INTERFACE I_HostOutputPorts EXTENDS __SYSTEM.IQueryInterface

METHOD PUBLIC AddDataAsOutputPort : I_OutputPort
VAR_INPUT
	Name : T_MAXSTRING;
	Data : I_Datatype;
END_VAR
END_METHOD

METHOD AddOutputPort
VAR_INPUT
	OutputPort : I_OutputPort;
END_VAR
END_METHOD

METHOD PUBLIC TryGetOutputPortByName : BOOL
VAR_INPUT
	Name : T_MAXSTRING;
	Destination : REFERENCE TO I_OutputPort;
END_VAR
END_METHOD

END_INTERFACE

(* stored: Version 1.1.0.1, ProductVersion 3.1.4024.12
   Itf I_HostOutputPorts: Id {5e1aea97-5e53-08af-11e9-4031292affee}
   Method AddDataAsOutputPort: Id {ae2495e6-ec41-49e7-bdb1-5ba1eea57cfd}
   Method AddOutputPort: Id {ccc39ff5-e25c-0f20-3efe-f937f75d1bdc}
   Method TryGetOutputPortByName: Id {a3a67671-970b-01d6-2705-151b345eba16} *)
